PROGRAM Comp01_Devices
VAR
	Step_0: Step;
END_VAR

Lifts();
Servos();

ACTION Conveyors:
// NETWORK 1
END_ACTION

ACTION ConveyorStops:
// NETWORK 1
END_ACTION

ACTION LiftAndTransfers:
// NETWORK 1
END_ACTION

ACTION Lifts:
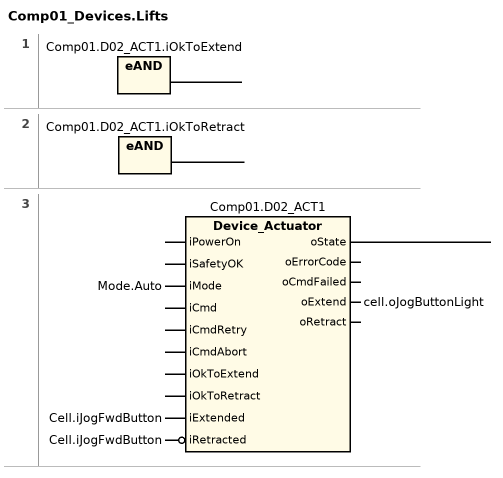
// NETWORK 1
Comp01.D02_ACT1.iOkToExtend(); // eAND

// NETWORK 2
Comp01.D02_ACT1.iOkToRetract(); // eAND

// NETWORK 3
Comp01.D02_ACT1(
    iMode := Mode.Auto,
    iExtended := Cell.iJogFwdButton,
    iRetracted := NOT Cell.iJogFwdButton,
    oExtend => cell.oJogButtonLight); // Device_Actuator
END_ACTION

ACTION Servos:
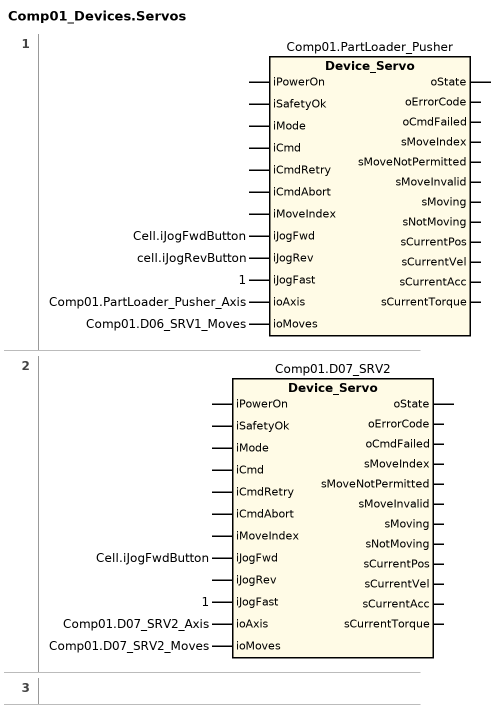
// NETWORK 1
Comp01.PartLoader_Pusher(
    iJogFwd := Cell.iJogFwdButton,
    iJogRev := cell.iJogRevButton,
    iJogFast := 1,
    ioAxis := Comp01.PartLoader_Pusher_Axis,
    ioMoves := Comp01.D06_SRV1_Moves); // Device_Servo

// NETWORK 2
Comp01.D07_SRV2(
    iJogFwd := Cell.iJogFwdButton,
    iJogFast := 1,
    ioAxis := Comp01.D07_SRV2_Axis,
    ioMoves := Comp01.D07_SRV2_Moves); // Device_Servo

// NETWORK 3
END_ACTION

END_PROGRAM

(* stored: Version 1.1.0.1, ProductVersion 3.1.4022.11
   POU Comp01_Devices: Id {f0a046c5-ec80-4bdc-848e-27d048afa24d}, SpecialFunc None
   Action Conveyors: Id {384c999c-2d61-41f6-9f17-2222a9754f90}
   Action ConveyorStops: Id {eb60ca93-9cce-4862-bfb3-f8780b314574}
   Action LiftAndTransfers: Id {265a0ec8-3a9e-4581-8aed-237c71a00e30}
   Action Lifts: Id {6d8a1d68-4091-4119-9dcf-9feebf32806f}
   Action Servos: Id {dfa8bfe5-7073-4b59-a3cb-a32e24979de3} *)
